// TIA Portal project "Chapa_GF1" (V14)

(* hardware
DEVICE "S7-1200 station_1"  S7-1200 Station
   slot 0: "Rack_0"  S7-1200 Rack  Rack  V1.0
   slot 1: "PLC_Publisher"  CPU 1211C DC/DC/DC  6ES7 211-1AE40-0XB0  V4.2
*)

// ===== PLC "PLC_Publisher"  CPU 1211C DC/DC/DC =====

VAR_GLOBAL   // PLC tag table "Tabla de variables estándar"
   "EntradaBotonAveria1" AT %I0.0 : Bool;
   "LEDAveria1" AT %Q0.0 : Bool;
   "Fallo Ciclo B1" AT %M100.0 : Bool;
END_VAR

TYPE "typeTcpConnParam"
VERSION : 0.1
   STRUCT
      hwIdentifier : Hw_Any;
      connectionID : Conn_Ouc;
      ipAdressBroker : Array[0..3] of Byte;
      localPort : UInt;
      mqttPort : UInt := 0;
   END_STRUCT;
END_TYPE

TYPE "typeMqttParam"
   STRUCT
      connectFlag : "typeMqttConnectFlags";
      publishFlag : "typeMqttPublishFlags";
      keepAlive : Word := 16#0A;
      packetIdentifier : Word := 16#10;
      clientIdentifier : String[23];   // should be PROFINET devicename
      willTopic : String[100];
      willMessage : String[100];
      userName : String[20];   // must be set, if flag "username" is true
      password : String[20];   // must be set, if flag "password" is true
      topic : String[100];
      message : String;
   END_STRUCT;
END_TYPE

TYPE "typeMqttConnectFlags"
   STRUCT
      cleanSession : Bool;
      will : Bool;
      willQoS_1 : Bool;   // true, if QoS = 1
      willQoS_2 : Bool;   // true, if QoS = 2
      willRetain : Bool;   // must be false, if Will flag is false
      password : Bool;   // if true, a password is required
      userName : Bool;   // if true, a username is required
   END_STRUCT;
END_TYPE

TYPE "typeMqttPublishFlags"
   STRUCT
      qualityOfService : Int;   // could be 0, 1, 2
      retain : Bool;
   END_STRUCT;
END_TYPE

TYPE "tipoPilaEnvio"
   STRUCT
      Zona : String;
      Elemento : String;
      Nombre_Averia : String;
      Valor_Averia : String;
   END_STRUCT;
END_TYPE

// folder: EnvioAveriasFijo

DATA_BLOCK "LMqtt_Publisher_DB"   // DB1
{ S7_Optimized_Access := 'TRUE' }
VERSION : 0.1
// stored: InstanceOfName LMqtt_Publisher
"LMqtt_Publisher"
BEGIN
END_DATA_BLOCK

DATA_BLOCK "LMqtt_Data"   // DB4
{ S7_Optimized_Access := 'TRUE' }
VERSION : 0.1
   VAR
      dataTcp : "typeTcpConnParam";
      dataMqtt : "typeMqttParam";
   END_VAR
BEGIN
   dataMqtt.password := 'asdf1234';
   dataMqtt.userName := 'eduardo';
   dataMqtt.connectFlag.userName := TRUE;
   dataMqtt.connectFlag.password := TRUE;
   dataMqtt.keepAlive := 16#003C;
   dataMqtt.publishFlag.qualityOfService := 2;
   dataMqtt.message := '0';
   dataTcp.hwIdentifier := 64;
   dataTcp.connectionID := 16#0002;
   dataTcp.ipAdressBroker[0] := 16#C0;
   dataMqtt.topic := 'Averias/Nave Pintura/Transportadores/GF15/Zona 1/CR1/B2';
   dataMqtt.willMessage := '1';
   dataMqtt.willTopic := 'Averias/Nave Pintura/Transportadores/GF15//Conexion';
   dataMqtt.clientIdentifier := 'publicadorPLC';
   dataTcp.localPort := 2000;
   dataTcp.mqttPort := 1883;
   dataMqtt.connectFlag.willRetain := TRUE;
   dataMqtt.connectFlag.willQoS_1 := FALSE;
   dataMqtt.connectFlag.will := TRUE;
   dataMqtt.connectFlag.cleanSession := TRUE;
   dataTcp.ipAdressBroker[1] := 16#A8;
   dataTcp.ipAdressBroker[2] := 16#01;
   dataTcp.ipAdressBroker[3] := 16#1E;
   dataMqtt.connectFlag.willQoS_2 := TRUE;
   dataMqtt.publishFlag.retain := TRUE;
   dataMqtt.packetIdentifier := 16#0010;
END_DATA_BLOCK

DATA_BLOCK "PilaEnvios"   // DB9
{ S7_Optimized_Access := 'TRUE' }
VERSION : 0.1
   VAR
      Puntero : Int := 1;
      N_Max_Registros : Int := 10;
      Averias_Enviar : Array[1..10] of "tipoPilaEnvio";
   END_VAR
BEGIN
END_DATA_BLOCK

DATA_BLOCK "VariablesEnvio"   // DB12
{ S7_Optimized_Access := 'TRUE' }
VERSION : 0.1
   VAR
      HabilitarMQTT : Bool;
      PublicarMQTT : Bool;
      TCPOk : Bool;
      MQTTOk : Bool;
      MQTTTrabajando : Bool;
      MQTTError : Bool;
      MQTTStatus : DWord;
      MQTTStatusID : Int;
      FP_HabilitarMQTT : Bool;
   END_VAR
BEGIN
END_DATA_BLOCK

// folder: EnvioAveriasVariable

DATA_BLOCK "ConfigEnviosAverias"   // DB8
{ S7_Optimized_Access := 'TRUE' }
VERSION : 0.1
   VAR
      Area : String := 'Chapa';
      Subarea : String := 'Transportadores';
      Sistema : String := 'GF1';
      ip_server : Array[0..3] of Byte;
      Usuario : String := 'eduardo';
      password : String := 'asdf1234';
   END_VAR
BEGIN
   ip_server[0] := 192;
   ip_server[1] := 168;
   ip_server[2] := 1;
   ip_server[3] := 30;
END_DATA_BLOCK

DATA_BLOCK "Flancos"   // DB11
{ S7_Optimized_Access := 'TRUE' }
VERSION : 0.1
   VAR
      "CR1 Cota 0 Fallo Ciclo B1 1" : Bool;
      "CR1 Cota 0 Fallo Ciclo B1 0" : Bool;
      "CR1 Mqtt Mqtt Conexion 0" : Bool;
      FlancoBoton1_0 : Bool;
      FlancoBoton1_1 : Bool;
   END_VAR
BEGIN
END_DATA_BLOCK

// folder: System blocks/Program resources

DATA_BLOCK "IEC_Timer_0_DB_HabilitarMQTT"   // DB10
{ S7_Optimized_Access := 'TRUE' }
AUTHOR : Simatic
FAMILY : IEC
NAME : IEC_TMR
VERSION : 1.0
// stored: InstanceOfName IEC_TIMER
"IEC_TIMER"
BEGIN
END_DATA_BLOCK

// folder: (top level)

ORGANIZATION_BLOCK "Main"   // OB1, LAD, ProgramCycle
TITLE = "Main Program Sweep (Cycle)" / Bloque Principal (OB1)
{ S7_Optimized_Access := 'TRUE' }
VERSION : 0.1
   VAR_INPUT
      Initial_Call : Bool;   // Initial call of this OB
      Remanence : Bool;   // =True, if remanent data are available
   END_VAR
   VAR_TEMP   // added for the SCL form of the ladder/FBD networks
      _w1 : Bool;
      _w2 : Bool;
   END_VAR
BEGIN

REGION Network 1: Llamada al bloque inicial del manejador de envios de averias
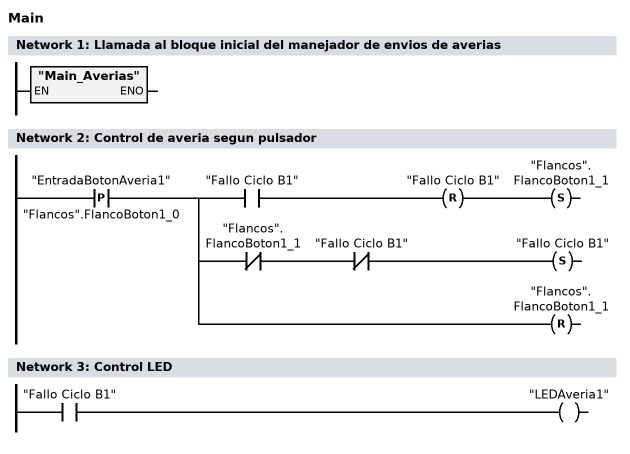
   RUNG wire#powerrail
      "Main_Averias"()
   END_RUNG
   // the same network as SCL:
   "Main_Averias"();
END_REGION

REGION Network 2: Control de averia segun pulsador
   RUNG wire#powerrail
      P_Contact(operand := "EntradaBotonAveria1", bit := "Flancos".FlancoBoton1_0)
      wire#w1
      Contact( "Fallo Ciclo B1" )
      R_Coil( "Fallo Ciclo B1" )
      S_Coil( "Flancos".FlancoBoton1_1 )
   END_RUNG
   RUNG wire#w1
      I_Contact( "Flancos".FlancoBoton1_1 )
      I_Contact( "Fallo Ciclo B1" )
      S_Coil( "Fallo Ciclo B1" )
   END_RUNG
   RUNG wire#w1
      R_Coil( "Flancos".FlancoBoton1_1 )
   END_RUNG
   // the same network as SCL:
   #_w1 := "EntradaBotonAveria1" AND NOT "Flancos".FlancoBoton1_0;   // rising edge of "EntradaBotonAveria1"
   "Flancos".FlancoBoton1_0 := "EntradaBotonAveria1";
   #_w2 := #_w1 AND "Fallo Ciclo B1";
   IF #_w2 THEN
       "Fallo Ciclo B1" := FALSE;
       "Flancos".FlancoBoton1_1 := TRUE;
   END_IF;
   IF #_w1 AND NOT "Flancos".FlancoBoton1_1 AND NOT "Fallo Ciclo B1" THEN "Fallo Ciclo B1" := TRUE; END_IF;
   IF #_w1 THEN "Flancos".FlancoBoton1_1 := FALSE; END_IF;
END_REGION

REGION Network 3: Control LED
   RUNG wire#powerrail
      Contact( "Fallo Ciclo B1" )
      Coil( "LEDAveria1" )
   END_RUNG
   // the same network as SCL:
   "LEDAveria1" := "Fallo Ciclo B1";
END_REGION
END_ORGANIZATION_BLOCK

// folder: EnvioAveriasFijo

FUNCTION_BLOCK "LMqtt_Publisher"   // FB2, SCL
{ S7_Optimized_Access := 'TRUE' }
VERSION : 0.1
   VAR_INPUT
      enable : Bool;
      publish : Bool;
      tcpConnParam : "typeTcpConnParam";
      mqttParam : "typeMqttParam";
   END_VAR
   VAR_OUTPUT
      tcpEstablished : Bool;
      mqttEstablished : Bool;
      published : Bool;
      busy : Bool;
      error : Bool;
      status : DWord;
      statusID : Int;
   END_VAR
   VAR
      statTcpConnParam : TCON_IP_v4;
      instTcpConnect : TCON;
      instTcpSend : TSEND;
      instTcpRCV : TRCV;
      instTcpDisconnect : TDISCON;
      instWatchDog : TON_TIME;
      instKeepAlive : TON_TIME;
      statStateMQTT : Int;
      statStateMQTTinternal : Int;
      statStateTCP : Int;
      statLastState : Int;
      statConnectLenght : Int;
      statCorrectOffset : Int;
      statSendLenght : Int;
      statConnectEncodedLenght : Int;
      statConnectLenghtOffset : Int;
      statKeepAliveTime : Time;
      statI : Int;
      statPacketID : Word;
      statPacketIDAck : Word;
      statRcvLen : UDInt;
      statPublishOld : Bool;
      statReConnect : Bool;
      statEnableOld : Bool;
      statMqttResetOld : Bool;
      statTriggerWatchDog : Bool;
      statTriggerKeepAlive : Bool;
      statNewDataRcv : Bool;
      statKeepAliveOff : Bool;
      statSendBuffer : Array[1..1000] of Byte;
      statRcvBuffer : Array[1..200] of Byte;
   END_VAR
   VAR_TEMP
      tempStringToChar : Array[0..255] of Char;
      tempCountChars : UInt;
      tempLenght : Word;
   END_VAR
   VAR CONSTANT
      TCP_PARAM : Int := 1;
      TCP_DISCONNECT : Int := -1;
      TCP_ERROR : Int := -2;
      TCP_CONNECTED : Int := 3;
      TCP_CONNECTING : Int := 2;
      MQTT_CONNECT_FLAG_CHECK : Int := 10;
      MQTT_CONNECT : Int := 11;
      MQTT_PUBLISH : Int := 13;
      MQTT_DISCONNECT : Int := 15;
      MQTT_CONNACK : Int := 12;
      MQTT_PUBACK : Int := 14;
      MQTT_PING : Int := 17;
      MQTT_PINGRESP : Int := 18;
      MQTT_PUBREL : Int := 19;
      MQTT_PUBCOMP : Int := 20;
      MQTT_IDLE : Int;
      MQTT_CONNECTED : Int := 16;
      MQTT_DISCONNECTED : Int := -11;
      MQTT_ERROR : Int := -12;
      IDLE : Int;
      TIME_MONITORING : Int := 20;
      WATCHDOG_TIME : Time := t#30s;
      MQTT_MSG_TYPE_CONNACK : Int := 32;
      MQTT_MSG_TYPE_DISCONNECT : Int := 224;
      MQTT_MSG_TYPE_PUBACK : Int := 64;
      MQTT_MSG_TYPE_PUBREC : Int := 80;
      MQTT_MSG_TYPE_PUBCOM : Int := 112;
      MQTT_MSG_TYPE_PING : Int := 192;
      MQTT_MSG_TYPE_PINGRESP : Int := 208;
      MQTT_CONNACK_ACCEPTED : Int;
      MQTT_PORT : Word := 16#22B3;
      MQTT_PROTOCOL_NAME : String := 'MQTT';
      MQTT_ERROR_WILL_FLAG : Word := 16#80F0;
      MQTT_ERROR_QOS_FLAG : Word := 16#80F1;
      MQTT_ERROR_PACKETID : Word := 16#80F2;
      MQTT_ERROR_KEEPALIVE : Word := 16#80F3;
   END_VAR
   // statTcpConnParam.ActiveEstablished := true;
BEGIN
   //=============================================================================
   //SIEMENES AG
   //(c)Copyright 2016 All Rights Reserved
   //-----------------------------------------------------------------------------
   //Library:       (that the source is dedicated to)
   //Tested with:   (target system with FW Version)
   //Engineering:   TIA Portal V14
   //Restrictions:  (OB types, etc.)
   //Requirements:  (hardware, technological package, memory needed, etc.)
   //Functionality: MQTT
   //-----------------------------------------------------------------------------
   //Change log table:
   //Version  Date       Expert in charge Changes applied
   //01.00.00 dd.mm.yyyy (name of expert) First released version
   //=============================================================================
   //Establish TCP Connection to be ready for MQTT

   IF #enable
       AND NOT #statEnableOld
   THEN
       #statStateTCP := #TCP_PARAM;
       #statStateMQTT := #MQTT_DISCONNECTED;
       #instWatchDog.IN := false;
       #statPublishOld := #publish;
   END_IF;

   IF NOT #enable
       AND #statEnableOld
   THEN
       IF #error = 1
       THEN
           #statStateTCP := #IDLE;
           #error := 0;
       ELSE
           #statStateMQTT := #MQTT_DISCONNECT;
           //#statStateTCP := #TCP_DISCONNECT;
       END_IF;
   END_IF;

    #instWatchDog(IN := #statTriggerWatchDog,PT := #WATCHDOG_TIME);

   REGION State maschine TCP
       CASE #statStateTCP OF
           #IDLE:
               IF NOT #error
               THEN
                   #status := 0;
                   #statusID := 0;
                   #error := 0;
                   #statTcpConnParam.ID := #tcpConnParam.connectionID;
                   #instTcpDisconnect(ID := #statTcpConnParam.ID);
                   #instTcpConnect(ID := #statTcpConnParam.ID,
                                   CONNECT := #statTcpConnParam);
               END_IF;
               #published := 0;
               #busy := false;
               #mqttEstablished := false;
               #statMqttResetOld := 0;
               #tcpEstablished := false;
               #statStateMQTT := #MQTT_DISCONNECTED;
               #statStateMQTTinternal := #IDLE;
               #statTriggerWatchDog := false;
               #statTriggerKeepAlive := 0;
               IF #statLastState=#TCP_DISCONNECT
               THEN
                   #error := 0;
                   END_IF;
           #TCP_CONNECTED:
               ;
               //Check TCP Connection
               IF #instTcpRCV.STATUS > w#16#80C0
               THEN
                   #statStateTCP := #TCP_ERROR;
                   #statusID := #TCP_CONNECTED;
               END_IF;

           #TCP_PARAM:
               #statTcpConnParam.InterfaceId := #tcpConnParam.hwIdentifier;
               #statTcpConnParam.ID := #tcpConnParam.connectionID;
               #statTcpConnParam.LocalPort := #tcpConnParam.localPort;
               #statTcpConnParam.RemotePort := #tcpConnParam.mqttPort;
               #statTcpConnParam.RemoteAddress.ADDR[1] := #tcpConnParam.ipAdressBroker[0];
               #statTcpConnParam.RemoteAddress.ADDR[2] := #tcpConnParam.ipAdressBroker[1];
               #statTcpConnParam.RemoteAddress.ADDR[3] := #tcpConnParam.ipAdressBroker[2];
               #statTcpConnParam.RemoteAddress.ADDR[4] := #tcpConnParam.ipAdressBroker[3];

             #statStateTCP := #TCP_CONNECTING;
           #TCP_CONNECTING:
               REGION TCP Connect
                   #statTriggerWatchDog := true;
                   #instTcpConnect.REQ := NOT #instTcpConnect.REQ XOR #instTcpConnect.BUSY;
                   #instTcpConnect(ID := #statTcpConnParam.ID,
                                   CONNECT := #statTcpConnParam);

                   IF (#instTcpConnect.DONE)
                       AND (#instTcpConnect.BUSY = 0)
                       AND (#instTcpConnect.REQ)
                   THEN
                       #instTcpConnect.REQ := false;
                       #tcpEstablished := true;
                       #statStateTCP := #TCP_CONNECTED;
                       #statTriggerWatchDog := false;
                   ELSIF (#instTcpConnect.ERROR)
                   THEN
                       #statusID := #TCP_CONNECTING;
                       #instTcpConnect.REQ := false;
                       #statStateTCP := #TCP_ERROR;
                   END_IF;
               END_REGION

           #TCP_DISCONNECT:
               REGION TCP Disconnect
                   #instTcpDisconnect.REQ := NOT #instTcpDisconnect.REQ XOR #instTcpDisconnect.BUSY;
                   #statTriggerWatchDog := false;
                   #instTcpDisconnect(ID := #statTcpConnParam.ID);

                   IF (#instTcpDisconnect.DONE)
                   THEN
                       //Done with success
                       #instTcpDisconnect.REQ := false;
                       #statLastState := #TCP_DISCONNECT;
                       #statStateTCP := #IDLE;
                   ELSIF (#instTcpDisconnect.ERROR)
                   THEN
                       #statusID := #TCP_DISCONNECT;
                       #instTcpDisconnect.REQ := false;
                       #statStateTCP := #TCP_ERROR;
                   END_IF;
               END_REGION
               ;
           #TCP_ERROR:
               REGION Errorhandling
                   #error := true;
                   #statStateMQTT := #MQTT_DISCONNECTED;
                   #statStateMQTTinternal := #IDLE;
                   #tcpEstablished := false;
                   #mqttEstablished := false;
                   #published := false;
                   #statTriggerWatchDog := false;
                       CASE #statusID OF
                           #TCP_CONNECTING:
                               #statStateTCP := #IDLE;
                               #status := #instTcpConnect.STATUS;
                           #TCP_CONNECTED:
                               #statStateTCP := #TCP_DISCONNECT;
                               #status := #instTcpRCV.STATUS;
                           #TCP_DISCONNECT:
                               //pointless for a retry at TDISCON
                               #statStateTCP := #IDLE;
                               #status := #instTcpDisconnect.STATUS;
                           #TIME_MONITORING:
                               #statStateTCP := #TCP_DISCONNECT;
                               #status := T_CONV(IN := #instWatchDog.ET);
                           ELSE
                               ;
                       END_CASE;
               END_REGION
               ;
           ELSE
               ;
       END_CASE;
   END_REGION
   #statEnableOld := #enable;
   REGION WatchDog
       IF #instWatchDog.Q = true
       THEN
           #statStateTCP := #TCP_ERROR;
           #statusID := #TIME_MONITORING;
       END_IF;
   END_REGION

   REGION OUC blocks

       #instTcpSend(ID:=#statTcpConnParam.ID,
                     DATA:=#statSendBuffer);
        #instTcpRCV(EN_R:=true,
                    ID:=#statTcpConnParam.ID,
                   LEN:=0,
                   ADHOC:=1,
                   RCVD_LEN=>#statRcvLen,
                   DATA:=#statRcvBuffer);
       IF #instTcpRCV.RCVD_LEN > 0 THEN
           #statNewDataRcv := 1;
       END_IF;

   END_REGION

   //Bring Statemachine in a definded state, if TCP Connection breaks
   IF #statStateMQTT > 0 AND
       #statStateTCP <> #TCP_CONNECTED
   THEN
       #statStateMQTT := #MQTT_DISCONNECTED;
       #instTcpSend.REQ := 0;
   END_IF;

   //MQTT makes no sense without an established TCP
   IF NOT (#statStateTCP = #TCP_CONNECTED)
   THEN
       RETURN;
   END_IF;




    #instKeepAlive(IN := #statTriggerKeepAlive,
                   PT := #statKeepAliveTime);
       CASE #statStateMQTT OF
           #MQTT_DISCONNECTED:
               #mqttEstablished := false;
               #statPublishOld := #publish;
               #statStateMQTT := #MQTT_CONNECT_FLAG_CHECK;
               #statStateMQTTinternal := #IDLE;
               #statTriggerKeepAlive := 0;
               #statKeepAliveOff := false;
               #statPacketID := #mqttParam.packetIdentifier;

           #MQTT_CONNECT_FLAG_CHECK:
               #busy := 1;
               //validate flags
               IF #mqttParam.connectFlag.willRetain
                   AND NOT #mqttParam.connectFlag.will
               THEN
                   #statStateMQTT := #MQTT_ERROR;
                   #statusID := #MQTT_CONNECT_FLAG_CHECK;
                   #status := #MQTT_ERROR_WILL_FLAG;
               ELSE
                   IF NOT #mqttParam.connectFlag.will
                       AND (#mqttParam.connectFlag.willQoS_1 OR #mqttParam.connectFlag.willQoS_2)
                   THEN
                       #statStateMQTT := #MQTT_ERROR;
                       #statusID := #MQTT_CONNECT_FLAG_CHECK;
                       #status := #MQTT_ERROR_QOS_FLAG;
                   ELSE
                       IF (#mqttParam.connectFlag.willQoS_1
                           AND #mqttParam.connectFlag.willQoS_2)
                       THEN
                           #statStateMQTT := #MQTT_ERROR;
                           #statusID := #MQTT_CONNECT_FLAG_CHECK;
                           #status := #MQTT_ERROR_QOS_FLAG;
                       ELSE;
                        #statStateMQTT := #MQTT_CONNECT;
                       END_IF;
                   END_IF;

               END_IF;
               IF (WORD_TO_INT(#mqttParam.keepAlive) = 0)
               THEN
                   #statKeepAliveOff := true;
               END_IF;
               IF (WORD_TO_INT(#mqttParam.keepAlive) < 2)
                   AND
                   (WORD_TO_INT(#mqttParam.keepAlive) > 0)
               THEN
                   #statStateMQTT := #MQTT_ERROR;
                   #statusID := #MQTT_CONNECT_FLAG_CHECK;
                   #status := #MQTT_ERROR_KEEPALIVE;
               END_IF;
               IF (WORD_TO_INT(#mqttParam.keepAlive) > 2)
               THEN
                   #statKeepAliveOff := false;
               END_IF;
           #MQTT_CONNECT:
                REGION MQTT Connect

                   //Calculate Remaining Lenght
                   #statConnectLenght := 10 + LEN(IN := #mqttParam.clientIdentifier) + 2;
                   IF #mqttParam.connectFlag.userName
                   THEN
                       #statConnectLenght := #statConnectLenght + LEN(IN := #mqttParam.userName) + 2;
                   END_IF;
                   IF #mqttParam.connectFlag.password
                   THEN
                       #statConnectLenght := #statConnectLenght + LEN(IN := #mqttParam.password) + 2;
                   END_IF;
                   IF #mqttParam.connectFlag.will
                   THEN
                       #statConnectLenght := #statConnectLenght + LEN(IN := #mqttParam.willMessage) + LEN(IN := #mqttParam.willTopic) + 4;
                   END_IF;
                   #statConnectLenghtOffset := 0;
                   //Build Telegram
                   //Fixed Header
                   #statSendBuffer[1] := 16#10;

                   #statSendLenght :=#statConnectLenght;
                   WHILE (#statConnectLenght > 0)
                   DO
                       #statConnectEncodedLenght := #statConnectLenght MOD 128;
                       #statConnectLenght := #statConnectLenght / 128;
                       // if there are more data to encode, set the top bit of this byte
                       IF #statConnectLenght > 0
                       THEN
                           #statConnectEncodedLenght := #statConnectEncodedLenght OR 128;
                           #statSendBuffer[2 + #statConnectLenghtOffset] := INT_TO_BYTE(#statConnectEncodedLenght);
                           #statConnectLenghtOffset := #statConnectLenghtOffset + 1;
                       ELSE
                           #statSendBuffer[2 + #statConnectLenghtOffset] := INT_TO_BYTE(#statConnectEncodedLenght);
                       END_IF;
                   END_WHILE;
                   #statSendLenght := #statSendLenght + #statConnectLenghtOffset;
                   //Variable Header
                   //Protocol name
                   #statSendBuffer[3 + #statConnectLenghtOffset] := 0;
                   #statSendBuffer[4 + #statConnectLenghtOffset] := 4;
                   #statSendBuffer[5 + #statConnectLenghtOffset] := 'M';
                   #statSendBuffer[6 + #statConnectLenghtOffset] := 'Q';
                   #statSendBuffer[7 + #statConnectLenghtOffset] := 'T';
                   #statSendBuffer[8 + #statConnectLenghtOffset] := 'T';
                   //Protocol Level
                   #statSendBuffer[9 + #statConnectLenghtOffset] := 4;
                   //Connect Flags
                   #statSendBuffer[10 + #statConnectLenghtOffset].%X0 := 0;
                   #statSendBuffer[10 + #statConnectLenghtOffset].%X1 := #mqttParam.connectFlag.cleanSession;
                   #statSendBuffer[10 + #statConnectLenghtOffset].%X2 := #mqttParam.connectFlag.will;
                   #statSendBuffer[10 + #statConnectLenghtOffset].%X3 := #mqttParam.connectFlag.willQoS_1;
                   #statSendBuffer[10 + #statConnectLenghtOffset].%X4 := #mqttParam.connectFlag.willQoS_2;
                   #statSendBuffer[10 + #statConnectLenghtOffset].%X5 := #mqttParam.connectFlag.willRetain;
                   #statSendBuffer[10 + #statConnectLenghtOffset].%X6 := #mqttParam.connectFlag.password;
                   #statSendBuffer[10 + #statConnectLenghtOffset].%X7 := #mqttParam.connectFlag.userName;
                   //Keep Alive in sec
                  #statSendBuffer[11 + #statConnectLenghtOffset] := #mqttParam.keepAlive.%B1;
                  #statSendBuffer[12 + #statConnectLenghtOffset] := #mqttParam.keepAlive.%B0;
                   //Payload
                   //ClientIdentifier
                   #tempLenght := INT_TO_WORD(LEN(IN := #mqttParam.clientIdentifier));
                   #statSendBuffer[13 + #statConnectLenghtOffset] := #tempLenght.%B1;
                   #statSendBuffer[14 + #statConnectLenghtOffset] := #tempLenght.%B0;
                   Strg_TO_Chars(Strg := #mqttParam.clientIdentifier,
                                 pChars := 0,
                                 Cnt => #tempCountChars,
                                 Chars := #tempStringToChar);
                   FOR #statI := 0 TO UINT_TO_INT(#tempCountChars - 1) DO
                       #statSendBuffer[15 + #statConnectLenghtOffset + #statI] := #tempStringToChar[#statI];
                   END_FOR;
                   #statConnectLenghtOffset := #statConnectLenghtOffset + #statI;
                   //WillTopic and WillMessage
                   IF #mqttParam.connectFlag.will THEN
                       #statCorrectOffset := 0;
                       #tempLenght:=INT_TO_WORD(LEN(IN := #mqttParam.willTopic));
                       #statSendBuffer[15 + #statConnectLenghtOffset] := #tempLenght.%B1;
                       #statSendBuffer[16 + #statConnectLenghtOffset] := #tempLenght.%B0;
                       Strg_TO_Chars(Strg := #mqttParam.willTopic,
                                     pChars := 0,
                                     Cnt => #tempCountChars,
                                     Chars := #tempStringToChar);
                       FOR #statI := 0 TO UINT_TO_INT(#tempCountChars - 1) DO
                           #statSendBuffer[17 + #statConnectLenghtOffset + #statI] := #tempStringToChar[#statI];
                       END_FOR;
                       #statConnectLenghtOffset := #statConnectLenghtOffset + #statI;

                       #tempLenght:=INT_TO_WORD(LEN(IN := #mqttParam.willMessage));
                       #statSendBuffer[17 + #statConnectLenghtOffset] := #tempLenght.%B1;
                       #statSendBuffer[18 + #statConnectLenghtOffset] := #tempLenght.%B0;
                       Strg_TO_Chars(Strg := #mqttParam.willMessage,
                                     pChars := 0,
                                     Cnt => #tempCountChars,
                                     Chars := #tempStringToChar);
                       FOR #statI := 0 TO UINT_TO_INT(#tempCountChars - 1) DO
                           #statSendBuffer[19 + #statConnectLenghtOffset + #statI] := #tempStringToChar[#statI];
                       END_FOR;
                       #statConnectLenghtOffset := #statConnectLenghtOffset + #statI;
                   ELSE
                       #statCorrectOffset := 4;
                   END_IF;
                   //UserName
                   IF #mqttParam.connectFlag.userName THEN
                       #tempLenght := INT_TO_WORD(LEN(IN := #mqttParam.userName));
                       #statSendBuffer[19 + #statConnectLenghtOffset - #statCorrectOffset] := #tempLenght.%B1;
                       #statSendBuffer[20 + #statConnectLenghtOffset - #statCorrectOffset] := #tempLenght.%B0;
                       Strg_TO_Chars(Strg := #mqttParam.userName,
                                     pChars := 0,
                                     Cnt => #tempCountChars,
                                     Chars := #tempStringToChar);
                       FOR #statI := 0 TO UINT_TO_INT(#tempCountChars - 1) DO
                           #statSendBuffer[21 + #statConnectLenghtOffset + #statI-#statCorrectOffset] := #tempStringToChar[#statI];
                       END_FOR;
                       #statConnectLenghtOffset := #statConnectLenghtOffset + #statI;
                   END_IF;
                   //Password
                   IF #mqttParam.connectFlag.password THEN
                       #tempLenght := INT_TO_WORD(LEN(IN := #mqttParam.password));
                       #statSendBuffer[21 + #statConnectLenghtOffset - #statCorrectOffset] := #tempLenght.%B1;
                       #statSendBuffer[22 + #statConnectLenghtOffset - #statCorrectOffset] := #tempLenght.%B0;
                       Strg_TO_Chars(Strg := #mqttParam.password,
                                     pChars := 0,
                                     Cnt => #tempCountChars,
                                     Chars := #tempStringToChar);
                       FOR #statI := 0 TO UINT_TO_INT(#tempCountChars - 1) DO
                           #statSendBuffer[23 + #statConnectLenghtOffset + #statI-#statCorrectOffset] := #tempStringToChar[#statI];
                       END_FOR;
                       #statConnectLenghtOffset := #statConnectLenghtOffset + #statI;
                   END_IF;

            #instTcpSend.REQ := true;
             #instTcpSend.LEN := INT_TO_UDINT(#statSendLenght + 2);

                   IF ((#instTcpSend.DONE)
                       AND (#instTcpSend.BUSY = 0))
                   THEN
                       #instTcpSend.REQ := false;
                       #statStateMQTT := #MQTT_CONNACK;
                       //Delete Send Buffer
                       FOR #statI := 1 TO (#statSendLenght + 2) DO
                           #statSendBuffer[#statI] := 0;
                       END_FOR;
                   ELSIF #instTcpSend.ERROR
                   THEN
                       #statusID := #MQTT_CONNECT;
                       #instTcpSend.REQ := false;
                       #statStateMQTT := #MQTT_ERROR;

                   END_IF;

               END_REGION
               ;
           #MQTT_CONNACK:
               IF #statNewDataRcv THEN

                   IF ((#statRcvBuffer[1] AND b#16#f0) = #MQTT_MSG_TYPE_CONNACK)
                       AND
                       (#statRcvBuffer[4] = #MQTT_CONNACK_ACCEPTED)
                   THEN
                       #statStateMQTT := #MQTT_CONNECTED;
                       #mqttEstablished := true;
                       #busy := false;
                       #statStateMQTTinternal := #IDLE;
                       //start Keep Alive Timer
                       //KeepAliveTImer is set to (Keep Alive (in s) - 2s)
                       #statKeepAliveTime := T_CONV((WORD_TO_UINT(#mqttParam.keepAlive) * 1000 - 2000));
                       IF NOT #statKeepAliveOff
                       THEN
                           #statTriggerKeepAlive := true;
                       END_IF;
                       #statNewDataRcv := 0;
                   ELSE
                       #statStateMQTT := #MQTT_ERROR;
                       #statusID := #MQTT_CONNACK;
                   END_IF;
               END_IF;
           #MQTT_CONNECTED:
               IF #publish
                   AND NOT #statPublishOld
                   AND (#statStateMQTTinternal=#IDLE)
               THEN
                   #statStateMQTTinternal := #MQTT_PUBLISH;
                   #published := 0;
                   #error := 0;
                  #statTriggerKeepAlive := false;
                   #statPacketID := #statPacketID + 1;
               END_IF;
               #statPublishOld := #publish;

                IF (#instKeepAlive.Q)
                    AND (#statStateMQTTinternal = #IDLE)
                    AND (NOT #statKeepAliveOff)
                THEN
                    #statStateMQTTinternal := #MQTT_PING;
                    #statTriggerKeepAlive := false;
                END_IF;
                CASE #statStateMQTTinternal OF
                    #IDLE:
                        #published := 0;
                        ;
                    #MQTT_PUBLISH:
                        ;
                        #busy := true;
                        #statConnectLenghtOffset := 0;
                        #statConnectLenght := LEN(IN := #mqttParam.topic) + LEN(IN := #mqttParam.message) + 2;
                        #statSendBuffer[1] := 16#30;
                        #statSendBuffer[1].%X0 := #mqttParam.publishFlag.retain;
                        #statSendBuffer[1].%X3 := false;
                        CASE #mqttParam.publishFlag.qualityOfService OF
                            0:
                                #statSendBuffer[1].%X1 := 0;
                                #statSendBuffer[1].%X2 := 0;
                            1:
                                #statSendBuffer[1].%X1 := 1;
                                #statSendBuffer[1].%X2 := 0;
                                //2 Byte Packet Identifiert added
                                #statConnectLenght := #statConnectLenght + 2;
                            2:
                                #statSendBuffer[1].%X1 := 0;
                                #statSendBuffer[1].%X2 := 1;
                                //2 Byte Packet Identifiert added
                                #statConnectLenght := #statConnectLenght + 2;
                            ELSE:
                                ;
                                #statStateMQTT := #MQTT_ERROR;
                                #statusID := #MQTT_PUBLISH;
                        END_CASE;
                        #statSendLenght := #statConnectLenght;
                        WHILE (#statConnectLenght > 0)
                        DO
                            #statConnectEncodedLenght := #statConnectLenght MOD 128;
                            #statConnectLenght := #statConnectLenght / 128;
                            // if there are more data to encode, set the top bit of this byte
                            IF #statConnectLenght > 0
                            THEN
                                #statConnectEncodedLenght := #statConnectEncodedLenght OR 128;
                                #statSendBuffer[2 + #statConnectLenghtOffset] := INT_TO_BYTE(#statConnectEncodedLenght);
                                #statConnectLenghtOffset := #statConnectLenghtOffset + 1;
                            ELSE
                                #statSendBuffer[2 + #statConnectLenghtOffset] := INT_TO_BYTE(#statConnectEncodedLenght);
                            END_IF;
                        END_WHILE;
                        #statSendLenght := #statSendLenght + #statConnectLenghtOffset;
                        //Variable Header
                        #tempLenght := INT_TO_WORD(LEN(IN := #mqttParam.topic));
                        #statSendBuffer[3 + #statConnectLenghtOffset] := #tempLenght.%B1;
                        #statSendBuffer[4 + #statConnectLenghtOffset] := #tempLenght.%B0;
                        Strg_TO_Chars(Strg := #mqttParam.topic,
                                      pChars := 0,
                                      Cnt => #tempCountChars,
                                      Chars := #tempStringToChar);
                        FOR #statI := 0 TO UINT_TO_INT(#tempCountChars - 1) DO
                            #statSendBuffer[5 + #statConnectLenghtOffset + #statI] := #tempStringToChar[#statI];
                        END_FOR;
                        #statConnectLenghtOffset := #statConnectLenghtOffset + #statI;
                        IF (#mqttParam.publishFlag.qualityOfService > 0)
                        THEN

                            #statSendBuffer[5 + #statConnectLenghtOffset] := #statPacketID.%B1;
                            #statSendBuffer[6 + #statConnectLenghtOffset] := #statPacketID.%B0;
                            //Payload
                            Strg_TO_Chars(Strg := #mqttParam.message,
                                          pChars := 0,
                                          Cnt => #tempCountChars,
                                          Chars := #tempStringToChar);
                            FOR #statI := 0 TO UINT_TO_INT(#tempCountChars - 1) DO
                                #statSendBuffer[7 + #statConnectLenghtOffset + #statI] := #tempStringToChar[#statI];
                            END_FOR;
                            #instTcpSend.LEN := INT_TO_UDINT(#statSendLenght + 2);
                        ELSE
                            Strg_TO_Chars(Strg := #mqttParam.message,
                                          pChars := 0,
                                          Cnt => #tempCountChars,
                                          Chars := #tempStringToChar);
                            FOR #statI := 0 TO UINT_TO_INT(#tempCountChars - 1) DO
                                #statSendBuffer[5 + #statConnectLenghtOffset + #statI] := #tempStringToChar[#statI];
                            END_FOR;
                            #instTcpSend.LEN := INT_TO_UDINT(#statSendLenght + 2);
                        END_IF;

                        #instTcpSend.REQ := true;


                        IF ((#instTcpSend.DONE)
                            AND (#instTcpSend.BUSY = 0))
                        THEN
                            #instTcpSend.REQ := false;
                            IF (#mqttParam.publishFlag.qualityOfService > 0)
                            THEN
                                #statPacketIDAck := #statPacketID;
                                #statStateMQTTinternal := #MQTT_PUBACK;
                            ELSE
                                //QoS = 0; finish here
                                #published := true;
                                #busy := false;
                                #statNewDataRcv := false;
                                IF NOT #statKeepAliveOff
                                THEN
                                    #statTriggerKeepAlive := true;
                                END_IF;

                                #statStateMQTTinternal := #IDLE;
                            END_IF;
                        ELSIF #instTcpSend.ERROR
                        THEN
                            #statusID := #MQTT_PUBLISH;
                            #instTcpSend.REQ := false;
                            #statStateMQTT := #MQTT_ERROR;
                            #status := #instTcpSend.STATUS;
                        END_IF;
                    #MQTT_PUBACK:
                        IF #statNewDataRcv THEN
                            IF ((#statRcvBuffer[1] AND b#16#f0) = #MQTT_MSG_TYPE_PUBACK)
                                OR
                                ((#statRcvBuffer[1] AND b#16#f0) = INT_TO_WORD(#MQTT_MSG_TYPE_PUBREC))
                            THEN
                                IF
                                    (#statRcvBuffer[3] = #statPacketIDAck.%B1)
                                    AND
                                    (#statRcvBuffer[4] = #statPacketIDAck.%B0)
                                THEN
                                    IF (#mqttParam.publishFlag.qualityOfService = 1)
                                    THEN
                                        //QoS = 1; finish here
                                        #statStateMQTTinternal := #MQTT_IDLE;
                                        #published := true;
                                        #busy := false;
                                        #statNewDataRcv := false;
                                        //Re-Activate Kepp Alive Timer
                                        IF NOT #statKeepAliveOff
                                        THEN
                                            #statTriggerKeepAlive := true;
                                        END_IF;

                                        #statStateMQTTinternal := #IDLE;
                                    ELSE
                                        #statStateMQTTinternal := #MQTT_PUBREL;
                                    END_IF;
                                ELSE
                                    #statNewDataRcv := false;
                                END_IF;
                            ELSE
                                #statStateMQTT := #MQTT_ERROR;
                                #statusID := #MQTT_PUBACK;
                            END_IF;
                        END_IF;
                    #MQTT_PUBREL:
                        //fixed Header
                        #statSendBuffer[1] := 16#62;
                        #statSendBuffer[2] := 2;
                        //Variable Header
                        #statSendBuffer[3] := #statPacketID.%B1;
                        #statSendBuffer[4] := #statPacketID.%B0;
                        #instTcpSend.LEN := INT_TO_UDINT(4);
                        #instTcpSend.REQ := true;

                        IF ((#instTcpSend.DONE)
                            AND (#instTcpSend.BUSY = 0))
                        THEN
                            #instTcpSend.REQ := false;
                            #statPacketIDAck := #statPacketID;
                            #statStateMQTTinternal := #MQTT_PUBCOMP;

                        ELSIF #instTcpSend.ERROR
                        THEN
                            #statusID := #MQTT_PUBREL;
                            #instTcpSend.REQ := false;
                            #statStateMQTT := #MQTT_ERROR;
                            #status := #instTcpSend.STATUS;
                        END_IF;
                    #MQTT_PUBCOMP:
                        IF #statNewDataRcv THEN
                            IF ((#statRcvBuffer[1] AND b#16#f0) = #MQTT_MSG_TYPE_PUBCOM)
                            THEN
                                IF
                                    (#statRcvBuffer[3] = #statPacketIDAck.%B1)
                                    AND
                                    (#statRcvBuffer[4] = #statPacketIDAck.%B0)
                                THEN
                                    //QoS = 2; finish here
                                    #statStateMQTTinternal := #MQTT_IDLE;
                                    #published := true;
                                    #busy := false;
                                    #statNewDataRcv := false;
                                    //Re-Activate Kepp Alive Timer
                                    IF NOT #statKeepAliveOff
                                    THEN
                                        #statTriggerKeepAlive := true;
                                    END_IF;

                                    #statStateMQTTinternal := #IDLE;
                                ELSE
                                    #statStateMQTT := #MQTT_ERROR;
                                    #statusID := #MQTT_PUBCOMP;
                                END_IF;
                            END_IF;
                        END_IF;
                    #MQTT_PING:

                        #busy := true;
                        //Build fixed Header
                        //Message Type
                        #statSendBuffer[1] := INT_TO_BYTE(#MQTT_MSG_TYPE_PING);
                        //Remaining Lenght (must be O)
                        #statSendBuffer[2] := 0;
                        #instTcpSend.REQ := true;
                        #instTcpSend.LEN := 2;

                        IF ((#instTcpSend.DONE)
                            AND (#instTcpSend.BUSY = 0))
                        THEN
                            #instTcpSend.REQ := false;
                            #statStateMQTTinternal := #MQTT_PINGRESP;
                        ELSIF #instTcpSend.ERROR
                        THEN
                            #statusID := #MQTT_PING;
                            #instTcpSend.REQ := false;
                            #statStateMQTT := #MQTT_ERROR;
                            #status := #instTcpSend.STATUS;
                        END_IF;
                    #MQTT_PINGRESP:
                        IF #statNewDataRcv
                        THEN
                            IF ((#statRcvBuffer[1] AND b#16#f0) = #MQTT_MSG_TYPE_PINGRESP)
                            THEN
                                #busy := false;
                                #statNewDataRcv := false;
                                #statTriggerKeepAlive := true;
                                #statStateMQTTinternal := #IDLE;
                            END_IF;
                        ELSE
                            #statNewDataRcv := false;
                        END_IF;

                END_CASE;
           #MQTT_DISCONNECT:
           #busy := 0;
           //Build fixed Header
           //Message Type
           #statSendBuffer[1] := INT_TO_BYTE(#MQTT_MSG_TYPE_DISCONNECT);
           //Remaining Lenght (must be O)
           #statSendBuffer[2] := 0;
           #instTcpSend.REQ := true;
           #instTcpSend.LEN := 2;

           IF ((#instTcpSend.DONE)
               AND (#instTcpSend.BUSY = 0))
           THEN
               IF NOT #enable THEN
                   #statStateTCP := #TCP_DISCONNECT;
               END_IF;
               #instTcpSend.REQ := false;
               #statStateMQTT := #MQTT_DISCONNECTED;
               #statStateMQTTinternal := #IDLE;
           ELSIF #instTcpSend.ERROR
           THEN
               IF NOT #enable THEN
                   #statStateTCP := #TCP_DISCONNECT;
               END_IF;
               #statusID := #MQTT_DISCONNECT;
               #instTcpSend.REQ := false;
               #statStateMQTT := #MQTT_ERROR;
               #status := #instTcpSend.STATUS;
           END_IF;
               #MQTT_ERROR:

               REGION Errorhandling MQTT
                   #error := true;
                   #busy := false;
                   #statStateMQTTinternal := #IDLE;
                   #statTriggerKeepAlive := 0;
                   #statKeepAliveOff := false;
                 CASE #statusID OF
                     #MQTT_CONNECT_FLAG_CHECK:
                         #mqttEstablished := false;
                         #statStateMQTT := #MQTT_DISCONNECTED;
                         ;
                     #MQTT_CONNECT:
                         #mqttEstablished := false;
                         #status := #instTcpSend.STATUS;   ;
                         #statStateMQTT := #MQTT_DISCONNECTED;
                       #MQTT_CONNACK:
                           #mqttEstablished := false;
                           #status := #statRcvBuffer[4];
                           #statStateMQTT := #MQTT_DISCONNECTED;
                       #MQTT_PUBLISH:
                               #published := false;
                               #statStateMQTT := #MQTT_CONNECTED;
                               #MQTT_PUBACK,#MQTT_PUBCOMP,#MQTT_PUBREL:
                           #published := false;
                           #status :=#MQTT_ERROR_PACKETID;
                           #statStateMQTT := #MQTT_CONNECTED;
                       #MQTT_PINGRESP:;
                           #MQTT_PING:;
                       #MQTT_DISCONNECT:
                           #mqttEstablished := false;
                          ;
                       ELSE
                           ;
                   END_CASE;
              END_REGION
               ;



       END_CASE
       ;
END_FUNCTION_BLOCK

FUNCTION "Main_MQTT" : Void   // FC1, SCL
{ S7_Optimized_Access := 'TRUE' }
VERSION : 0.1
   VAR_TEMP
      published : Bool;
      error : Bool;
      status : DWord;
      statusID : Int;
      tcpOK : Bool;
      mqttOK : Bool;
      reiniciar_conexion : Bool;
      done_TDISCON : Bool;
      busy_TDISCON : Bool;
      error_TDISCON : Bool;
      status_TDISCON : Word;
      Topic : String;
      i : Int;
      listo_para_envio : Bool;
   END_VAR
BEGIN
   //
   //Fichero:     Main_MAQTT
   // Version:     1.0
   // Autor:       Eduardo Buetas Sanjuan
   // Proyecto:    Trabajo investigacion de Evaluacion Continua
   // Asignatura:  Generacion Automatica de Codigo
   // Titulacion:  Master Universitario en Investigacion en Ingenieria de Software y Sistemas Informaticos.
   // Centro:      UNED
   // Fecha:       14/04/2018
   // Ejecutable:  No
   // Proposito:   Esta funcion se encarga de enviar por MQTT las averias incluidas en la pila de averias PilaEnvios
   //              para el envio de los datos a traves de MQTT se vale de la libreria LMqtt_Publisher publicado por Siemens AG
   //              como ejemplo de aplicacion en su pagina web y de los tipos de usuario y DB de datos del mismo ejemplo de 
   //              aplicacion. 
   //
   // Esta funcion forma parte de la fuente fija del generador de sistemas de envio de averias AVERIAS_MDA_S7_1200
   // No debe ser modificado de manera manual en ningun caso
   REGION envios mqtt

       "LMqtt_Publisher_DB"(enable := "VariablesEnvio".HabilitarMQTT,
                            publish := "VariablesEnvio".PublicarMQTT,
                            tcpConnParam := "LMqtt_Data".dataTcp,
                            mqttParam := "LMqtt_Data".dataMqtt,
                            tcpEstablished => "VariablesEnvio".TCPOk,
                            mqttEstablished => "VariablesEnvio".MQTTOk,
                            busy => "VariablesEnvio".MQTTTrabajando,
                            published => #published,
                            error => #error,
                            status => #status,
                            statusID => #statusID);

       IF "VariablesEnvio".MQTTOk AND NOT "VariablesEnvio".PublicarMQTT THEN
           #listo_para_envio := true;
       ELSE
           #listo_para_envio := false;
       END_IF;
       IF #published THEN
           //Como se ha publicado correctamente borramos el envio de la pila 
           "VariablesEnvio".PublicarMQTT := false;
           FOR #i := 1 TO "PilaEnvios".Puntero DO
               "PilaEnvios".Averias_Enviar[#i] := "PilaEnvios".Averias_Enviar[#i + 1];
           END_FOR;
           "PilaEnvios".Puntero := "PilaEnvios".Puntero - 1;
       END_IF;

       IF #error THEN
           IF #statusID = 2 AND #status = 16#80A3 THEN
               //si el error es que esta la id de conexion ocupada antes de reintentar la conexion desacemos esa conexion
               #reiniciar_conexion := true;
           END_IF;
           "VariablesEnvio".MQTTStatus := #status;
           "VariablesEnvio".MQTTStatusID := #statusID;
           "VariablesEnvio".MQTTError := #error;
           "VariablesEnvio".PublicarMQTT := false;
           "VariablesEnvio".HabilitarMQTT := false;
       END_IF;
       IF "VariablesEnvio".TCPOk AND "VariablesEnvio".MQTTOk THEN
           "VariablesEnvio".MQTTStatus := 0;
           "VariablesEnvio".MQTTStatusID := 0;
           "VariablesEnvio".MQTTError := FALSE;
       END_IF;

       "TDISCON_DB"(REQ := #reiniciar_conexion,
                    ID := "LMqtt_Data".dataTcp.connectionID,
                    DONE => #done_TDISCON,
                    BUSY => #busy_TDISCON,
                    ERROR => #error_TDISCON,
                    STATUS => #status_TDISCON);
   END_REGION
   REGION "Datos de conexion MQTT"
       //Datos fijos de conexion MQTT
       #Topic := 'Averias/';
       #Topic := CONCAT(IN1:=#Topic, IN2:="ConfigEnviosAverias".Area);
       #Topic := CONCAT(IN1 := #Topic, IN2 := '/');
       #Topic := CONCAT(IN1 := #Topic, IN2 := "ConfigEnviosAverias".Subarea);
       #Topic := CONCAT(IN1 := #Topic, IN2 := '/');
       #Topic := CONCAT(IN1 := #Topic, IN2 := "ConfigEnviosAverias".Sistema);
       #Topic := CONCAT(IN1 := #Topic, IN2 := '/');
       "LMqtt_Data".dataMqtt.userName := "ConfigEnviosAverias".Usuario; //usuario de conexion 
       "LMqtt_Data".dataMqtt.password := "ConfigEnviosAverias".password; //password de conexion 
       //Will topic se refiere al mensaje que se le enviara a los suscriptores en el caso de la perdida de conexion 
       //con el publicador, este mensaje se almacena en el broker hasta que el publicador pierde la conexion con el 
       //broker en este momento el mensaje es enviado a los suscriptores
       "LMqtt_Data".dataMqtt.willTopic := CONCAT(IN1 := #Topic, IN2 := 'Mqtt/Mqtt/Conexion');
       "LMqtt_Data".dataMqtt.willMessage := '1';
       "LMqtt_Data".dataMqtt.connectFlag.will := TRUE;
       "LMqtt_Data".dataMqtt.connectFlag.willQoS_1 := FALSE;
       "LMqtt_Data".dataMqtt.connectFlag.willQoS_2 := TRUE;
       "LMqtt_Data".dataMqtt.connectFlag.willRetain := true;
       //Los mensajes que envie este publicador se almacenaran en el broker hasta que todos los 
       //suscripotores los reciban
       "LMqtt_Data".dataMqtt.publishFlag.retain := true;
       //Los mensajes intercamebiados por este suscriptor con el broker se enviaran con una 
       //calidad deservicio QoS=2
       "LMqtt_Data".dataMqtt.publishFlag.qualityOfService := 2;
       //El timepo de KeepAlive sera de 60 segundos entre este publicador y el broker
       "LMqtt_Data".dataMqtt.keepAlive := 60;
   END_REGION
   REGION "habilitar conexion MQTT"
       //la conexion MQTT debe estar siempre habilitada, si no lo esta cada 30 segundos
       //se intentara la reconexion.

       "IEC_Timer_0_DB_HabilitarMQTT".TON(IN:=NOT "VariablesEnvio".HabilitarMQTT,
                                          PT:=T#30s,
                                          Q=>"VariablesEnvio".FP_HabilitarMQTT);
       IF "VariablesEnvio".FP_HabilitarMQTT THEN
           "VariablesEnvio".HabilitarMQTT := true;
      END_IF;

   END_REGION
   REGION Envio de mensajes de averia desde la pila
       //Estos datos son fijos para todos los envios por MQTT de las averias
       IF "PilaEnvios".Puntero > 1 AND #listo_para_envio THEN //si la pila es <> 1
                                                              //es que hay algo que enviar, si no se esta enviando se envia
           #Topic := CONCAT(IN1 := #Topic, IN2 := "PilaEnvios".Averias_Enviar[1].Zona);
           #Topic := CONCAT(IN1 := #Topic, IN2 := '/');
           #Topic:= CONCAT(IN1 := #Topic, IN2 :="PilaEnvios".Averias_Enviar[1].Elemento);
           #Topic := CONCAT(IN1 := #Topic, IN2 := '/');
           "LMqtt_Data".dataMqtt.topic := CONCAT(IN1 := #Topic, IN2 := "PilaEnvios".Averias_Enviar[1].Nombre_Averia);
           "LMqtt_Data".dataMqtt.message := "PilaEnvios".Averias_Enviar[1].Valor_Averia;
           "VariablesEnvio".PublicarMQTT:= true;
       END_IF;
   END_REGION
   // Esta funcion forma parte de la fuente fija del generador de sistemas de envio de averias AVERIAS_MDA_S7_1200
   // No debe ser modificado de manera manual en ningun caso
END_FUNCTION

// folder: EnvioAveriasVariable

FUNCTION "Main_Averias" : Void   // FC2, SCL
{ S7_Optimized_Access := 'TRUE' }
VERSION : 0.1
BEGIN
   (*
   * Control de envio de averias a traves de pila, se controlan dos averias 
   * Alarma 1: "Averias/Chapa/Transportadores/GF1/Cota 0/CR1/Fallo Ciclo B1"
   * Conexion: "Averias/Chapa/Transportadores/GF1/Mqtt/Mqtt/Conexion"
   * Este topico con el mensjae "1" se configurara para ser enviado cuando haya una
   * desconexion del sistema (opcion will conexion)
   * Cuando la averia en cuestion se active enviara un mensaje "1" y cuando la se resuelva
   * enviara un mensaje "0"
   * Los envios de mensajes siempre seranc on QoS=2 
   * Destinatario: Trabajo Fin de Master
   *               Master Investigacion en Ingenieria de Software y
   *               Sistemas Informaticos
   * Proyecto: Sistema de propagacion de averias en la Industria 4.0
   * Fecha Creacion: 11/05/2018
   * Fecha Revision: 11/05/2018
   * @author: Eduardo Buetas
   * @version: 1.0
   *)
   REGION Cota 0
       REGION Fallo Ciclo B1
           IF "Fallo Ciclo B1" AND NOT "Flancos"."CR1 Cota 0 Fallo Ciclo B1 1" THEN
               "PilaEnvios".Averias_Enviar["PilaEnvios".Puntero].Zona := 'Cota 0';
               "PilaEnvios".Averias_Enviar["PilaEnvios".Puntero].Elemento := 'CR1';
               "PilaEnvios".Averias_Enviar["PilaEnvios".Puntero].Nombre_Averia := 'Fallo Ciclo B1';
               "PilaEnvios".Averias_Enviar["PilaEnvios".Puntero].Valor_Averia := '1';
               "PilaEnvios".Puntero := "PilaEnvios".Puntero + 1;
               "Flancos"."CR1 Cota 0 Fallo Ciclo B1 1" := true;
           END_IF;
           IF NOT "Fallo Ciclo B1" THEN
               "Flancos"."CR1 Cota 0 Fallo Ciclo B1 1" := false;
           END_IF;
           IF NOT "Fallo Ciclo B1" AND NOT "Flancos"."CR1 Cota 0 Fallo Ciclo B1 0" THEN
               "PilaEnvios".Averias_Enviar["PilaEnvios".Puntero].Zona := 'Cota 0';
               "PilaEnvios".Averias_Enviar["PilaEnvios".Puntero].Elemento := 'CR1';
               "PilaEnvios".Averias_Enviar["PilaEnvios".Puntero].Nombre_Averia := 'Fallo Ciclo B1';
               "PilaEnvios".Averias_Enviar["PilaEnvios".Puntero].Valor_Averia := '0';
               "PilaEnvios".Puntero := "PilaEnvios".Puntero + 1;
               "Flancos"."CR1 Cota 0 Fallo Ciclo B1 0" := true;
           END_IF;
           IF "Fallo Ciclo B1" THEN
               "Flancos"."CR1 Cota 0 Fallo Ciclo B1 0" := false;
           END_IF;
       END_REGION
       REGION conexion
           IF "VariablesEnvio".MQTTOk AND NOT "Flancos"."CR1 Mqtt Mqtt Conexion 0" THEN
               "PilaEnvios".Averias_Enviar["PilaEnvios".Puntero].Zona := 'Mqtt';
               "PilaEnvios".Averias_Enviar["PilaEnvios".Puntero].Elemento := 'Mqtt';
               "PilaEnvios".Averias_Enviar["PilaEnvios".Puntero].Nombre_Averia := 'Conexion';
               "PilaEnvios".Averias_Enviar["PilaEnvios".Puntero].Valor_Averia := '0';
               "PilaEnvios".Puntero := "PilaEnvios".Puntero + 1;
               "Flancos"."CR1 Mqtt Mqtt Conexion 0" := true;
           END_IF;
           IF NOT "VariablesEnvio".MQTTOk THEN
               "Flancos"."CR1 Mqtt Mqtt Conexion 0" := false;
           END_IF;
       END_REGION
   END_REGION

   "Main_MQTT"(); //lamada a la funcion que envia las averias que mete este fichero en la pila de envio de averias.

   // Esta funcion forma parte de la fuente fija del generador de sistemas de envio de averias AVERIAS_MDA_S7_1200
   // No debe ser modificado de manera manual en ningun caso
END_FUNCTION